{attribute addProperty BoxType "EL3681-0000-0017"}
{attribute addProperty Id "UnderrangeBIT10.1251OverrangeBIT10.1252Extended_rangeBIT10.1253Data_InvalidBIT10.1254Range_InvalidBIT10.1255Autorange_enabledBIT10.1256ErrorBIT10.1257Calibration_in_progressBIT10.1258TxPDO_StateBIT10.1257TxPDO_ToggleBIT10.1259"}
{attribute addProperty CRC "1844918370"}
{attribute addProperty SizeInBites "16"}
{attribute addProperty SizeInBytes "2"}
TYPE Status_6DF73862 :
STRUCT
	{attribute addProperty Name "Underrange"}
	Underrange : BIT;
	{attribute addProperty Name "Overrange"}
	Overrange : BIT;
	{attribute addProperty Name "Extended_range"}
	Extended_range : BIT;
	{attribute addProperty Name "Data_Invalid"}
	Data_Invalid : BIT;
	{attribute addProperty Name "Range_Invalid"}
	Range_Invalid : BIT;
	{attribute addProperty Name "Autorange_enabled"}
	Autorange_enabled : BIT;
	{attribute addProperty Name "Error"}
	Error : BIT;
	{attribute addProperty Name "Calibration_in_progress"}
	Calibration_in_progress : BIT;
	{attribute 'hide'}
	reserve_1_BIT_0 : BIT;
	{attribute 'hide'}
	reserve_1_BIT_1 : BIT;
	{attribute 'hide'}
	reserve_1_BIT_2 : BIT;
	{attribute 'hide'}
	reserve_1_BIT_3 : BIT;
	{attribute 'hide'}
	reserve_1_BIT_4 : BIT;
	{attribute 'hide'}
	reserve_1_BIT_5 : BIT;
	{attribute addProperty Name "TxPDO_State"}
	TxPDO_State : BIT;
	{attribute addProperty Name "TxPDO_Toggle"}
	TxPDO_Toggle : BIT;
END_STRUCT
END_TYPE

(* stored: Version 1.2.0.0, ProductVersion 3.1.4024.9
   DUT Status_6DF73862: Id {28e98f78-ab10-481a-b464-1126e8b6b732} *)
